FUNCTION_BLOCK FB57
TITLE = 'fault'
AUTHOR : CB

VAR
	fault_F1 : FB45;
	fault_F2 : FB51;
	fault_F3 : FB55;
END_VAR


BEGIN


NETWORK
TITLE =
//
//	fault/fault_F1
CALL #fault_F1;



NETWORK
TITLE =
//
//	fault/fault_F2
CALL #fault_F2;



NETWORK
TITLE =
//
//	fault/fault_F3
CALL #fault_F3;




END_FUNCTION_BLOCK
